# EPICS autosave request: CARS/iocBoot/iocPINK/auto_settings.req
file "XFM_motor_settings.req",        P=XF:04BM-ES:2:, M=m1
file "XFM_motor_settings.req",        P=XF:04BM-ES:2:, M=m2
file "XFM_motor_settings.req",        P=XF:04BM-ES:2:, M=m3
